Universal Robots PolyScope program: forcabasic.urp

Program forcabasic (installation=default directory=/programs createdIn=5.9.3 lastSavedIn=5.14.5 robotSerialNumber=20195300809)
Calibrated DH parameters: a=[-0.000085, -0.20076, -0.212369, 0.000121, -0.000118, 0]; d=[0.15185, -26.306375, 24.753047, 1.684739, 0.085386, 0.092088]; alpha=[1.572149, -0.00522, -0.011864, 1.571339, -1.571085, 0]; deltaTheta=[0, 0.599885, -0.513355, -0.086555, 0.000006, 0]
InitVariablesNode
Robot Program (runOnlyOnce=false)
  Force Frame feature=Joint_6_name; selection=[0, 0, 1, 0, 0, 0]; wrench=[0, 0, 10, 0, 0, 0]; limitsForce=[0.15, 0.15, 0.005, 1.047198, 1.047198, 1.047198]; limitsMotion=[0.1, 0.1, 0.1, 0.349066, 0.349066, 0.349066]
    MoveJ speed 60 deg/s, acceleration 80 deg/s^2 (useActiveTCP=true) feature=Base
      Waypoint Waypoint_1: TCP in base x=154.261 y=-283.726 z=202.997 mm, rx=0.9545 ry=-2.9929 rz=0.0203 rad; joints [-37.465, -94.084, -57.724, -117.575, 89.069, 17.812] deg; TCP offset x=0 y=0 z=200 mm, rx=0 ry=0 rz=0 rad
      Waypoint Waypoint_2: TCP in base x=154.122 y=-283.644 z=132.042 mm, rx=0.9544 ry=-2.9929 rz=0.0199 rad; joints [-37.397, -88.674, -83.405, -97.317, 89.006, 17.647] deg
